/// This struct contains variables that
/// * are read from outside (e.g. HMI) to retrieve information about the unit's current state and (temporary) parameters (= `publish`) 
/// * are written from outside (e.g. HMI) to control the unit via ADS (= `subscribe`) 
TYPE TransportCom :
STRUCT
  Publish : TransportComPublish;
  Subscribe : TransportComSubscribe;
END_STRUCT
END_TYPE

(* stored: Version 1.1.0.1
   DUT TransportCom: Id {d7f3272d-b70b-406f-b5eb-b2b93d316afb} *)
